KUKA KRL data list: MathLibrary.dat

&ACCESS RVE
&REL 38
&PARAM EDITMASK = *
&PARAM TEMPLATE = C:\KRC\Roboter\Template\ExpertVorgabe
DEFDAT MathLibrary PUBLIC
  Global STRUC VECTOR3DTYPE REAL X,Y,Z
  Global STRUC ROTATIONSTYPE REAL A,B,C
  GLOBAL CONST REAL PI=3.1415926535897932384626433832795
ENDDAT
